{attribute 'GeneratedUsingTerminal: EP2328-1061-0016'}
{attribute addProperty BoxType "EP2328-1061-0016"}
{attribute addProperty Id "InputAT %I*BOOL1"}
{attribute addProperty CRC "2198356929"}
{attribute addProperty Size "1"}
TYPE DI_X02_Pin4_Input_830843C1 EXTENDS InputBase_8311D824 :
STRUCT
	{attribute addProperty Name "Input"}
	Input AT %I* : BOOL;
END_STRUCT
END_TYPE

(* stored: Version 1.2.0.0, ProductVersion 3.1.4024.9
   DUT DI_X02_Pin4_Input_830843C1: Id {49aecd53-cc91-400a-bc43-a83be971860c} *)
